(* PLC project parallel.project, CODESYS CODESYS V3.5 SP17 Patch 3 *)
(* stored: creationDateTime 2022-06-05T18:23:31.2070927, modificationDateTime 2022-05-14T22:34:49.5278322 *)

PROGRAM flow_1

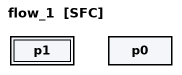
INITIAL_STEP p1:
END_STEP
STEP p0:
END_STEP
END_PROGRAM
